{attribute 'qualified_only'}
{attribute 'strict'}
{attribute 'to_string'}
TYPE E_MESSAGE_BATCH :
(
	MSG_BATCH_NULL,
  MSG_BATCH_JOB_STARTED,
  MSG_BATCH_NEXT_IN_JOB,
  MSG_BATCH_JOB_DONE
)UINT;
END_TYPE

(* stored: Version 1.1.0.1, ProductVersion 3.1.4026.20
   DUT E_MESSAGE_BATCH: Id {162dc715-735f-4446-b68a-d59bed78ed1b} *)
